Staubli VAL3: findItem.pgx

public program findItem(InstrItem x_iItem, num& x_nResult[], bool x_bUseSession)
// procedure
  local num i
  local num j
  local num l_nSize
  local string l_sProgName
  local bool l_bFound
  local num l_nSizeItem
  local InstrItem l_iItem
  local num z
  local string l_sSession
  local string l_sMessage
begin
  //
  // search in all of the program the x_iItem
  //
  call getSize(l_nSize)
  for i=0 to (l_nSize-1)
    // load all the program
    call get(l_sProgName,i)
    if l_sProgName!=""
      // SHOW THE program name
      call saveData:getSession(l_sSession)
      l_sMessage="SESSION:"+l_sSession+">SUB "+l_sProgName
      call use:typeLen(1,5,l_sMessage,38)
      // load the select program and search inside
      call load(l_sProgName,x_nResult)
      if x_nResult==0
        // SEARCH IN ALL THE ITEMS
        call getSizeItem(l_nSizeItem)
        if l_nSize!=0
          for j=0 to (l_nSizeItem-1)
            call getItem(l_iItem,j)
            // look inside
            l_bFound=(l_iItem.sType==x_iItem.sType and(l_iItem.sData==x_iItem.sData or find(l_iItem.sData," "+x_iItem.sData)!=-1))
            // use nested items
            if x_iItem.sType=="IN" or x_iItem.sType=="OUT" or x_iItem.sType=="NUM"
              l_bFound=l_bFound or (find(l_iItem.sData,x_iItem.sType)!=-1 and find(l_iItem.sData," "+x_iItem.sData)!=-1)
            else
              l_bFound=l_bFound or (find(l_iItem.sData,x_iItem.sType)!=-1 and find(l_iItem.sData+"#"," "+x_iItem.sData+"#")!=-1)
            endIf
            // FOUND IT
            if l_bFound
              x_nResult=-1
              call language:message(l_sMessage,23)
              popUpMsg(l_sMessage+x_iItem.sType+" "+x_iItem.sData+chr(10)+"SESSION:"+l_sSession+chr(10)+"SUB: "+l_sProgName+" > "+l_iItem.sType+" "+l_iItem.sData)
              // back
              return
            endIf
          endFor
        endIf
      else
        popUpMsg("error loading...SESSION:"+l_sSession+">SUB "+l_sProgName+" error "+toString("",x_nResult))
      endIf
    endIf
  endFor
end
